{attribute addProperty BoxType "EPP2038-0001-0016"}
{attribute addProperty Id "InputAT %I*BOOL81"}
{attribute addProperty CRC "3836671390"}
{attribute addProperty SizeInBites "8"}
{attribute addProperty SizeInBytes "1"}
TYPE Diag_Channel_E4AEF59E :
STRUCT
	{attribute addProperty Name "Input"}
	Input AT %I* : BOOL;
END_STRUCT
END_TYPE

(* stored: Version 1.2.0.0, ProductVersion 3.1.4024.9
   DUT Diag_Channel_E4AEF59E: Id {765523cb-9d39-46ee-b293-e264b19ef36c} *)
